{attribute 'pack_mode' := '1'}
TYPE ST_StatusNode :
STRUCT
	nState	: UINT;
	rTemp	: REAL;
END_STRUCT
END_TYPE

(* stored: Version 1.1.0.1, ProductVersion 3.1.4024.5
   DUT ST_StatusNode: Id {81872ef2-3d85-4d0d-a81f-9aeb2fd4db0d} *)
